LIN {X 0,Y 264.924,Z 479.026,A -85,B 0,C 180,E1 5571.318,E2 5571.318} C_VEL
LIN {X 0,Y 262.769,Z 475.669,A -85,B 0,C 180,E1 5567.921,E2 5567.921} C_VEL
LIN {X 0,Y 260.3,Z 472.231,A -85,B 0,C 180,E1 5561.41,E2 5561.41} C_VEL
LIN {X 0,Y 259.822,Z 472.519,A -85,B 0,C 180,E1 5558.558,E2 5558.558} C_VEL
LIN {X 0,Y 260.217,Z 475.555,A -85,B 0,C 180,E1 5552.295,E2 5552.295} C_VEL
LIN {X 0,Y 261.348,Z 479.248,A -85,B 0,C 180,E1 5548.559,E2 5548.559} C_VEL
LIN {X 0,Y 263.196,Z 484.586,A -85,B 0,C 180,E1 5544.765,E2 5544.765} C_VEL
LIN {X 0,Y 264.928,Z 489.758,A -85,B 0,C 180,E1 5542.035,E2 5542.035} C_VEL
LIN {X 0,Y 245.651,Z 644.406,A -85,B 0,C 180,E1 5539.399,E2 5539.399} C_VEL
LIN {X 0,Y 240.991,Z 667.184,A -85,B 0,C 180,E1 5538.834,E2 5538.834} C_VEL
LIN {X 0,Y 234.844,Z 688.807,A -85,B 0,C 180,E1 5538.055,E2 5538.055} C_VEL
LIN {X 0,Y 227.496,Z 709.005,A -85,B 0,C 180,E1 5537.061,E2 5537.061} C_VEL
LIN {X 0,Y 218.924,Z 728.293,A -85,B 0,C 180,E1 5535.814,E2 5535.814} C_VEL
LIN {X 0,Y 208.737,Z 747.497,A -85,B 0,C 180,E1 5534.186,E2 5534.186} C_VEL
LIN {X 0,Y 197.582,Z 765.406,A -85,B 0,C 180,E1 5532.183,E2 5532.183} C_VEL
LIN {X 0,Y 185.926,Z 781.624,A -85,B 0,C 180,E1 5529.792,E2 5529.792} C_VEL
LIN {X 0,Y 173.527,Z 796.762,A -85,B 0,C 180,E1 5526.82,E2 5526.82} C_VEL
LIN {X 0,Y 160.818,Z 810.467,A -85,B 0,C 180,E1 5523.174,E2 5523.174} C_VEL
LIN {X 0,Y 148.028,Z 822.753,A -85,B 0,C 180,E1 5518.662,E2 5518.662} C_VEL
LIN {X 0,Y 135.541,Z 833.645,A -85,B 0,C 180,E1 5513.019,E2 5513.019} C_VEL
LIN {X 0,Y 123.855,Z 843.086,A -85,B 0,C 180,E1 5505.936,E2 5505.936} C_VEL
LIN {X 0,Y 113.661,Z 850.993,A -85,B 0,C 180,E1 5497.079,E2 5497.079} C_VEL
LIN {X 0,Y 106.489,Z 856.756,A -85,B 0,C 180,E1 5487.315,E2 5487.315} C_VEL
LIN {X 0,Y 102.112,Z 860.954,A -85,B 0,C 180,E1 5476.414,E2 5476.414} C_VEL
LIN {X 0,Y 100.7,Z 863.459,A -85,B 0,C 180,E1 5465.36,E2 5465.36} C_VEL
LIN {X 0,Y 102.038,Z 864.682,A -85,B 0,C 180,E1 5453.997,E2 5453.997} C_VEL
LIN {X 0,Y 106.472,Z 864.54,A -85,B 0,C 180,E1 5442.914,E2 5442.914} C_VEL
LIN {X 0,Y 114.777,Z 862.689,A -85,B 0,C 180,E1 5432.097,E2 5432.097} C_VEL
LIN {X 0,Y 126.409,Z 858.943,A -85,B 0,C 180,E1 5422.802,E2 5422.802} C_VEL
LIN {X 0,Y 140.031,Z 853.547,A -85,B 0,C 180,E1 5415.453,E2 5415.453} C_VEL
LIN {X 0,Y 155.125,Z 846.474,A -85,B 0,C 180,E1 5409.569,E2 5409.569} C_VEL
LIN {X 0,Y 170.618,Z 838.065,A -85,B 0,C 180,E1 5405.018,E2 5405.018} C_VEL
LIN {X 0,Y 187.128,Z 827.692,A -85,B 0,C 180,E1 5401.224,E2 5401.224} C_VEL
LIN {X 0,Y 203.05,Z 816.054,A -85,B 0,C 180,E1 5398.276,E2 5398.276} C_VEL
LIN {X 0,Y 219.202,Z 802.456,A -85,B 0,C 180,E1 5395.814,E2 5395.814} C_VEL
LIN {X 0,Y 230.335,Z 791.931,A -85,B 0,C 180,E1 5394.32,E2 5394.32} C_VEL
LIN {X 0,Y 217.485,Z 805.371,A -85,B 0,C 180,E1 5392.785,E2 5392.785} C_VEL
LIN {X 0,Y 211.97,Z 810.64,A -85,B 0,C 180,E1 5392.344,E2 5392.344} C_VEL
LIN {X 0,Y 196.504,Z 823.434,A -85,B 0,C 180,E1 5391.994,E2 5391.994} C_VEL
LIN {X 0,Y 190.608,Z 828.015,A -85,B 0,C 180,E1 5391.411,E2 5391.411} C_VEL
LIN {X 0,Y 172.647,Z 841.576,A -85,B 0,C 180,E1 5388.143,E2 5388.143} C_VEL
LIN {X 0,Y 154.151,Z 853.984,A -85,B 0,C 180,E1 5383.715,E2 5383.715} C_VEL
LIN {X 0,Y 136.857,Z 864.412,A -85,B 0,C 180,E1 5378.088,E2 5378.088} C_VEL
LIN {X 0,Y 119.902,Z 873.894,A -85,B 0,C 180,E1 5370.13,E2 5370.13} C_VEL
LIN {X 0,Y 106.273,Z 881.294,A -85,B 0,C 180,E1 5360.223,E2 5360.223} C_VEL
LIN {X 0,Y 96.274,Z 886.967,A -85,B 0,C 180,E1 5347.78,E2 5347.78} C_VEL
LIN {X 0,Y 91.172,Z 890.787,A -85,B 0,C 180,E1 5333.932,E2 5333.932} C_VEL
LIN {X 0,Y 90.418,Z 892.658,A -85,B 0,C 180,E1 5322.122,E2 5322.122} C_VEL
LIN {X 0,Y 91.401,Z 893.227,A -85,B 0,C 180,E1 5312.501,E2 5312.501} C_VEL
LIN {X 0,Y 91.492,Z 893.013,A -85,B 0,C 180,E1 5308.115,E2 5308.115} C_VEL
LIN {X 0,Y 90.677,Z 891.796,A -85,B 0,C 180,E1 5299.832,E2 5299.832} C_VEL
LIN {X 0,Y 90.991,Z 889.004,A -85,B 0,C 180,E1 5288.732,E2 5288.732} C_VEL
LIN {X 0,Y 94.671,Z 884.089,A -85,B 0,C 180,E1 5275.954,E2 5275.954} C_VEL
LIN {X 0,Y 102.103,Z 877.465,A -85,B 0,C 180,E1 5264.36,E2 5264.36} C_VEL
LIN {X 0,Y 112.661,Z 868.974,A -85,B 0,C 180,E1 5254.612,E2 5254.612} C_VEL
LIN {X 0,Y 125.433,Z 858.784,A -85,B 0,C 180,E1 5246.767,E2 5246.767} C_VEL
LIN {X 0,Y 139.021,Z 847.405,A -85,B 0,C 180,E1 5240.766,E2 5240.766} C_VEL
LIN {X 0,Y 152.982,Z 834.686,A -85,B 0,C 180,E1 5236.092,E2 5236.092} C_VEL
LIN {X 0,Y 166.885,Z 820.612,A -85,B 0,C 180,E1 5232.41,E2 5232.41} C_VEL
LIN {X 0,Y 181.361,Z 804.213,A -85,B 0,C 180,E1 5229.289,E2 5229.289} C_VEL
LIN {X 0,Y 194.407,Z 787.495,A -85,B 0,C 180,E1 5226.945,E2 5226.945} C_VEL
LIN {X 0,Y 206.775,Z 769.259,A -85,B 0,C 180,E1 5225.031,E2 5225.031} C_VEL
LIN {X 0,Y 217.89,Z 750.129,A -85,B 0,C 180,E1 5223.53,E2 5223.53} C_VEL
LIN {X 0,Y 227.761,Z 730.153,A -85,B 0,C 180,E1 5222.336,E2 5222.336} C_VEL
LIN {X 0,Y 236.047,Z 710.089,A -85,B 0,C 180,E1 5221.423,E2 5221.423} C_VEL
LIN {X 0,Y 243.124,Z 688.824,A -85,B 0,C 180,E1 5220.708,E2 5220.708} C_VEL
LIN {X 0,Y 248.536,Z 667.243,A -85,B 0,C 180,E1 5220.164,E2 5220.164} C_VEL
LIN {X 0,Y 252.392,Z 644.573,A -85,B 0,C 180,E1 5219.681,E2 5219.681} C_VEL
LIN {X 0,Y 268.872,Z 495.81,A -85,B 0,C 180,E1 5217.075,E2 5217.075} C_VEL
LIN {X 0,Y 265.37,Z 489.707,A -85,B 0,C 180,E1 5213.293,E2 5213.293} C_VEL
LIN {X 0,Y 263.21,Z 486.145,A -85,B 0,C 180,E1 5210.379,E2 5210.379} C_VEL
LIN {X 0,Y 261.553,Z 483.485,A -85,B 0,C 180,E1 5207.64,E2 5207.64} C_VEL
LIN {X 0,Y 259.228,Z 480.152,A -85,B 0,C 180,E1 5201.33,E2 5201.33} C_VEL
LIN {X 0,Y 258.771,Z 480.458,A -85,B 0,C 180,E1 5198.626,E2 5198.626} C_VEL
LIN {X 0,Y 259.064,Z 483.366,A -85,B 0,C 180,E1 5192.588,E2 5192.588} C_VEL
LIN {X 0,Y 260.111,Z 487.05,A -85,B 0,C 180,E1 5188.869,E2 5188.869} C_VEL
LIN {X 0,Y 261.88,Z 492.466,A -85,B 0,C 180,E1 5185.063,E2 5185.063} C_VEL
LIN {X 0,Y 262.658,Z 495.183,A -85,B 0,C 180,E1 5183.653,E2 5183.653} C_VEL
LIN {X 0,Y 243.721,Z 644.757,A -85,B 0,C 180,E1 5181.215,E2 5181.215} C_VEL
LIN {X 0,Y 238.965,Z 667.665,A -85,B 0,C 180,E1 5180.679,E2 5180.679} C_VEL
LIN {X 0,Y 232.82,Z 688.959,A -85,B 0,C 180,E1 5179.955,E2 5179.955} C_VEL
LIN {X 0,Y 225.732,Z 708.262,A -85,B 0,C 180,E1 5179.066,E2 5179.066} C_VEL
LIN {X 0,Y 217.008,Z 727.792,A -85,B 0,C 180,E1 5177.889,E2 5177.889} C_VEL
LIN {X 0,Y 206.604,Z 747.209,A -85,B 0,C 180,E1 5176.348,E2 5176.348} C_VEL
LIN {X 0,Y 195.457,Z 764.898,A -85,B 0,C 180,E1 5174.497,E2 5174.497} C_VEL
LIN {X 0,Y 183.8,Z 780.948,A -85,B 0,C 180,E1 5172.285,E2 5172.285} C_VEL
LIN {X 0,Y 170.429,Z 796.941,A -85,B 0,C 180,E1 5169.321,E2 5169.321} C_VEL
LIN {X 0,Y 156.454,Z 811.547,A -85,B 0,C 180,E1 5165.564,E2 5165.564} C_VEL
LIN {X 0,Y 143.158,Z 823.823,A -85,B 0,C 180,E1 5161.125,E2 5161.125} C_VEL
LIN {X 0,Y 130.079,Z 834.717,A -85,B 0,C 180,E1 5155.501,E2 5155.501} C_VEL
LIN {X 0,Y 117.721,Z 844.169,A -85,B 0,C 180,E1 5148.321,E2 5148.321} C_VEL
LIN {X 0,Y 106.822,Z 852.097,A -85,B 0,C 180,E1 5139.161,E2 5139.161} C_VEL
LIN {X 0,Y 99.005,Z 857.931,A -85,B 0,C 180,E1 5128.749,E2 5128.749} C_VEL
LIN {X 0,Y 94.293,Z 862.111,A -85,B 0,C 180,E1 5117.14,E2 5117.14} C_VEL
LIN {X 0,Y 92.784,Z 864.707,A -85,B 0,C 180,E1 5104.844,E2 5104.844} C_VEL
LIN {X 0,Y 94.523,Z 865.971,A -85,B 0,C 180,E1 5092.164,E2 5092.164} C_VEL
LIN {X 0,Y 100.084,Z 865.743,A -85,B 0,C 180,E1 5079.724,E2 5079.724} C_VEL
LIN {X 0,Y 109.422,Z 863.853,A -85,B 0,C 180,E1 5068.705,E2 5068.705} C_VEL
LIN {X 0,Y 122.723,Z 859.924,A -85,B 0,C 180,E1 5059.093,E2 5059.093} C_VEL
LIN {X 0,Y 138.062,Z 854.158,A -85,B 0,C 180,E1 5051.698,E2 5051.698} C_VEL
LIN {X 0,Y 153.872,Z 847.013,A -85,B 0,C 180,E1 5046.222,E2 5046.222} C_VEL
LIN {X 0,Y 171.044,Z 837.891,A -85,B 0,C 180,E1 5041.755,E2 5041.755} C_VEL
LIN {X 0,Y 188.042,Z 827.35,A -85,B 0,C 180,E1 5038.317,E2 5038.317} C_VEL
LIN {X 0,Y 204.551,Z 815.529,A -85,B 0,C 180,E1 5035.637,E2 5035.637} C_VEL
LIN {X 0,Y 212.569,Z 809.08,A -85,B 0,C 180,E1 5034.476,E2 5034.476} C_VEL
LIN {X 0,Y 194.827,Z 824.66,A -85,B 0,C 180,E1 5032.062,E2 5032.062} C_VEL
LIN {X 0,Y 190.608,Z 828.015,A -85,B 0,C 180,E1 5031.411,E2 5031.411} C_VEL
LIN {X 0,Y 184.613,Z 832.571,A -85,B 0,C 180,E1 5030.763,E2 5030.763} C_VEL
LIN {X 0,Y 167.913,Z 843.389,A -85,B 0,C 180,E1 5029.908,E2 5029.908} C_VEL
LIN {X 0,Y 161.675,Z 847.223,A -85,B 0,C 180,E1 5029.028,E2 5029.028} C_VEL
LIN {X 0,Y 143.216,Z 858.371,A -85,B 0,C 180,E1 5024.441,E2 5024.441} C_VEL
LIN {X 0,Y 125.798,Z 867.854,A -85,B 0,C 180,E1 5018.409,E2 5018.409} C_VEL
LIN {X 0,Y 108.839,Z 876.387,A -85,B 0,C 180,E1 5009.704,E2 5009.704} C_VEL
LIN {X 0,Y 95.154,Z 883.089,A -85,B 0,C 180,E1 4998.24,E2 4998.24} C_VEL
LIN {X 0,Y 86.048,Z 887.879,A -85,B 0,C 180,E1 4983.892,E2 4983.892} C_VEL
LIN {X 0,Y 82.521,Z 890.822,A -85,B 0,C 180,E1 4968.355,E2 4968.355} C_VEL
LIN {X 0,Y 82.917,Z 891.818,A -85,B 0,C 180,E1 4956.919,E2 4956.919} C_VEL
LIN {X 0,Y 83.645,Z 891.917,A -85,B 0,C 180,E1 4950.678,E2 4950.678} C_VEL
LIN {X 0,Y 83.244,Z 891.408,A -85,B 0,C 180,E1 4945.17,E2 4945.17} C_VEL
LIN {X 0,Y 82.619,Z 889.427,A -85,B 0,C 180,E1 4933.831,E2 4933.831} C_VEL
LIN {X 0,Y 84.837,Z 885.454,A -85,B 0,C 180,E1 4920.323,E2 4920.323} C_VEL
LIN {X 0,Y 91.208,Z 879.636,A -85,B 0,C 180,E1 4907.174,E2 4907.174} C_VEL
LIN {X 0,Y 101.336,Z 871.983,A -85,B 0,C 180,E1 4895.985,E2 4895.985} C_VEL
LIN {X 0,Y 113.698,Z 862.812,A -85,B 0,C 180,E1 4887.343,E2 4887.343} C_VEL
LIN {X 0,Y 128.049,Z 851.724,A -85,B 0,C 180,E1 4880.434,E2 4880.434} C_VEL
LIN {X 0,Y 142.121,Z 839.968,A -85,B 0,C 180,E1 4875.444,E2 4875.444} C_VEL
LIN {X 0,Y 157.053,Z 826.029,A -85,B 0,C 180,E1 4871.34,E2 4871.34} C_VEL
LIN {X 0,Y 171.251,Z 811.205,A -85,B 0,C 180,E1 4868.237,E2 4868.237} C_VEL
LIN {X 0,Y 184.915,Z 795.071,A -85,B 0,C 180,E1 4865.759,E2 4865.759} C_VEL
LIN {X 0,Y 197.893,Z 777.601,A -85,B 0,C 180,E1 4863.767,E2 4863.767} C_VEL
LIN {X 0,Y 210.125,Z 758.395,A -85,B 0,C 180,E1 4862.142,E2 4862.142} C_VEL
LIN {X 0,Y 220.505,Z 739.281,A -85,B 0,C 180,E1 4860.924,E2 4860.924} C_VEL
LIN {X 0,Y 229.975,Z 718.523,A -85,B 0,C 180,E1 4859.917,E2 4859.917} C_VEL
LIN {X 0,Y 237.749,Z 697.676,A -85,B 0,C 180,E1 4859.159,E2 4859.159} C_VEL
LIN {X 0,Y 244.16,Z 675.65,A -85,B 0,C 180,E1 4858.583,E2 4858.583} C_VEL
LIN {X 0,Y 248.634,Z 653.809,A -85,B 0,C 180,E1 4858.117,E2 4858.117} C_VEL
LIN {X 0,Y 252.545,Z 622.713,A -85,B 0,C 180,E1 4857.551,E2 4857.551} C_VEL
LIN {X 0,Y 266.177,Z 501.282,A -85,B 0,C 180,E1 4855.476,E2 4855.476} C_VEL
LIN {X 0,Y 262.802,Z 495.248,A -85,B 0,C 180,E1 4851.358,E2 4851.358} C_VEL
LIN {X 0,Y 260.324,Z 491.281,A -85,B 0,C 180,E1 4847.316,E2 4847.316} C_VEL
LIN {X 0,Y 258.108,Z 488.034,A -85,B 0,C 180,E1 4841.011,E2 4841.011} C_VEL
LIN {X 0,Y 257.674,Z 488.539,A -85,B 0,C 180,E1 4838.37,E2 4838.37} C_VEL
LIN {X 0,Y 257.936,Z 491.276,A -85,B 0,C 180,E1 4832.781,E2 4832.781} C_VEL
LIN {X 0,Y 258.868,Z 494.803,A -85,B 0,C 180,E1 4829.219,E2 4829.219} C_VEL
LIN {X 0,Y 260.591,Z 500.432,A -85,B 0,C 180,E1 4825.307,E2 4825.307} C_VEL
LIN {X 0,Y 242.039,Z 645.097,A -85,B 0,C 180,E1 4823.058,E2 4823.058} C_VEL
LIN {X 0,Y 237.236,Z 667.943,A -85,B 0,C 180,E1 4822.557,E2 4822.557} C_VEL
LIN {X 0,Y 231.001,Z 689.276,A -85,B 0,C 180,E1 4821.88,E2 4821.88} C_VEL
LIN {X 0,Y 223.75,Z 708.751,A -85,B 0,C 180,E1 4821.039,E2 4821.039} C_VEL
LIN {X 0,Y 214.918,Z 728.218,A -85,B 0,C 180,E1 4819.937,E2 4819.937} C_VEL
LIN {X 0,Y 204.311,Z 747.686,A -85,B 0,C 180,E1 4818.486,E2 4818.486} C_VEL
LIN {X 0,Y 192.923,Z 765.427,A -85,B 0,C 180,E1 4816.737,E2 4816.737} C_VEL
LIN {X 0,Y 180.826,Z 781.713,A -85,B 0,C 180,E1 4814.61,E2 4814.61} C_VEL
LIN {X 0,Y 167.663,Z 797.067,A -85,B 0,C 180,E1 4811.91,E2 4811.91} C_VEL
LIN {X 0,Y 154.039,Z 810.974,A -85,B 0,C 180,E1 4808.549,E2 4808.549} C_VEL
LIN {X 0,Y 140.15,Z 823.513,A -85,B 0,C 180,E1 4804.31,E2 4804.31} C_VEL
LIN {X 0,Y 126.344,Z 834.65,A -85,B 0,C 180,E1 4798.87,E2 4798.87} C_VEL
LIN {X 0,Y 113.768,Z 843.888,A -85,B 0,C 180,E1 4792.21,E2 4792.21} C_VEL
LIN {X 0,Y 102.276,Z 851.801,A -85,B 0,C 180,E1 4783.575,E2 4783.575} C_VEL
LIN {X 0,Y 92.852,Z 858.206,A -85,B 0,C 180,E1 4772.475,E2 4772.475} C_VEL
LIN {X 0,Y 87.076,Z 862.639,A -85,B 0,C 180,E1 4760.089,E2 4760.089} C_VEL
LIN {X 0,Y 84.882,Z 865.617,A -85,B 0,C 180,E1 4746.398,E2 4746.398} C_VEL
LIN {X 0,Y 86.311,Z 867.154,A -85,B 0,C 180,E1 4732.968,E2 4732.968} C_VEL
LIN {X 0,Y 92.123,Z 867.233,A -85,B 0,C 180,E1 4719.01,E2 4719.01} C_VEL
LIN {X 0,Y 102.131,Z 865.538,A -85,B 0,C 180,E1 4707.029,E2 4707.029} C_VEL
LIN {X 0,Y 114.93,Z 862.236,A -85,B 0,C 180,E1 4697.725,E2 4697.725} C_VEL
LIN {X 0,Y 130.963,Z 856.914,A -85,B 0,C 180,E1 4690.009,E2 4690.009} C_VEL
LIN {X 0,Y 147.407,Z 850.224,A -85,B 0,C 180,E1 4684.43,E2 4684.43} C_VEL
LIN {X 0,Y 165.041,Z 841.662,A -85,B 0,C 180,E1 4679.999,E2 4679.999} C_VEL
LIN {X 0,Y 183.309,Z 831.088,A -85,B 0,C 180,E1 4676.471,E2 4676.471} C_VEL
LIN {X 0,Y 194.812,Z 823.518,A -85,B 0,C 180,E1 4674.64,E2 4674.64} C_VEL
LIN {X 0,Y 176.42,Z 837.275,A -85,B 0,C 180,E1 4671.853,E2 4671.853} C_VEL
LIN {X 0,Y 161.675,Z 847.223,A -85,B 0,C 180,E1 4669.028,E2 4669.028} C_VEL
LIN {X 0,Y 155.355,Z 850.938,A -85,B 0,C 180,E1 4668.048,E2 4668.048} C_VEL
LIN {X 0,Y 137.751,Z 859.678,A -85,B 0,C 180,E1 4666.353,E2 4666.353} C_VEL
LIN {X 0,Y 131.433,Z 862.733,A -85,B 0,C 180,E1 4664.999,E2 4664.999} C_VEL
LIN {X 0,Y 113.155,Z 871.566,A -85,B 0,C 180,E1 4658.078,E2 4658.078} C_VEL
LIN {X 0,Y 96.2,Z 879.117,A -85,B 0,C 180,E1 4647.988,E2 4647.988} C_VEL
LIN {X 0,Y 83.559,Z 884.671,A -85,B 0,C 180,E1 4634.899,E2 4634.899} C_VEL
LIN {X 0,Y 76.237,Z 888.317,A -85,B 0,C 180,E1 4619.02,E2 4619.02} C_VEL
LIN {X 0,Y 74.53,Z 890.286,A -85,B 0,C 180,E1 4603.175,E2 4603.175} C_VEL
LIN {X 0,Y 75.67,Z 890.639,A -85,B 0,C 180,E1 4591.506,E2 4591.506} C_VEL
LIN {X 0,Y 75.533,Z 890.311,A -85,B 0,C 180,E1 4586.957,E2 4586.957} C_VEL
LIN {X 0,Y 74.687,Z 888.722,A -85,B 0,C 180,E1 4576.048,E2 4576.048} C_VEL
LIN {X 0,Y 76.508,Z 885.109,A -85,B 0,C 180,E1 4561.075,E2 4561.075} C_VEL
LIN {X 0,Y 82.494,Z 879.907,A -85,B 0,C 180,E1 4547.245,E2 4547.245} C_VEL
LIN {X 0,Y 92.817,Z 872.605,A -85,B 0,C 180,E1 4535.035,E2 4535.035} C_VEL
LIN {X 0,Y 106.281,Z 863.376,A -85,B 0,C 180,E1 4525.415,E2 4525.415} C_VEL
LIN {X 0,Y 121.138,Z 852.652,A -85,B 0,C 180,E1 4518.328,E2 4518.328} C_VEL
LIN {X 0,Y 136.519,Z 840.416,A -85,B 0,C 180,E1 4513.057,E2 4513.057} C_VEL
LIN {X 0,Y 151.599,Z 826.97,A -85,B 0,C 180,E1 4509.109,E2 4509.109} C_VEL
LIN {X 0,Y 166.886,Z 811.628,A -85,B 0,C 180,E1 4505.958,E2 4505.958} C_VEL
LIN {X 0,Y 181.009,Z 795.521,A -85,B 0,C 180,E1 4503.57,E2 4503.57} C_VEL
LIN {X 0,Y 194.56,Z 777.741,A -85,B 0,C 180,E1 4501.644,E2 4501.644} C_VEL
LIN {X 0,Y 205.98,Z 760.302,A -85,B 0,C 180,E1 4500.233,E2 4500.233} C_VEL
LIN {X 0,Y 217.008,Z 740.709,A -85,B 0,C 180,E1 4499.033,E2 4499.033} C_VEL
LIN {X 0,Y 226.095,Z 721.625,A -85,B 0,C 180,E1 4498.138,E2 4498.138} C_VEL
LIN {X 0,Y 234.215,Z 700.744,A -85,B 0,C 180,E1 4497.404,E2 4497.404} C_VEL
LIN {X 0,Y 240.74,Z 679.476,A -85,B 0,C 180,E1 4496.864,E2 4496.864} C_VEL
LIN {X 0,Y 245.801,Z 656.965,A -85,B 0,C 180,E1 4496.402,E2 4496.402} C_VEL
LIN {X 0,Y 249.185,Z 633.378,A -85,B 0,C 180,E1 4495.971,E2 4495.971} C_VEL
LIN {X 0,Y 263.696,Z 507.078,A -85,B 0,C 180,E1 4493.906,E2 4493.906} C_VEL
LIN {X 0,Y 260.835,Z 501.998,A -85,B 0,C 180,E1 4490.068,E2 4490.068} C_VEL
LIN {X 0,Y 259.142,Z 499.12,A -85,B 0,C 180,E1 4487.07,E2 4487.07} C_VEL
LIN {X 0,Y 257.04,Z 495.955,A -85,B 0,C 180,E1 4480.929,E2 4480.929} C_VEL
LIN {X 0,Y 256.6,Z 496.55,A -85,B 0,C 180,E1 4478.275,E2 4478.275} C_VEL
LIN {X 0,Y 256.802,Z 499.085,A -85,B 0,C 180,E1 4473.08,E2 4473.08} C_VEL
LIN {X 0,Y 257.635,Z 502.557,A -85,B 0,C 180,E1 4469.573,E2 4469.573} C_VEL
LIN {X 0,Y 258.592,Z 506.364,A -85,B 0,C 180,E1 4466.959,E2 4466.959} C_VEL
LIN {X 0,Y 240.541,Z 645.36,A -85,B 0,C 180,E1 4464.923,E2 4464.923} C_VEL
LIN {X 0,Y 235.666,Z 668.296,A -85,B 0,C 180,E1 4464.457,E2 4464.457} C_VEL
LIN {X 0,Y 229.201,Z 690.109,A -85,B 0,C 180,E1 4463.811,E2 4463.811} C_VEL
LIN {X 0,Y 221.604,Z 710.096,A -85,B 0,C 180,E1 4463.001,E2 4463.001} C_VEL
LIN {X 0,Y 212.569,Z 729.539,A -85,B 0,C 180,E1 4461.964,E2 4461.964} C_VEL
LIN {X 0,Y 201.832,Z 748.804,A -85,B 0,C 180,E1 4460.611,E2 4460.611} C_VEL
LIN {X 0,Y 190.22,Z 766.486,A -85,B 0,C 180,E1 4458.967,E2 4458.967} C_VEL
LIN {X 0,Y 177.853,Z 782.736,A -85,B 0,C 180,E1 4456.961,E2 4456.961} C_VEL
LIN {X 0,Y 164.355,Z 798.084,A -85,B 0,C 180,E1 4454.4,E2 4454.4} C_VEL
LIN {X 0,Y 150.32,Z 811.981,A -85,B 0,C 180,E1 4451.19,E2 4451.19} C_VEL
LIN {X 0,Y 135.931,Z 824.521,A -85,B 0,C 180,E1 4447.102,E2 4447.102} C_VEL
LIN {X 0,Y 121.513,Z 835.67,A -85,B 0,C 180,E1 4441.783,E2 4441.783} C_VEL
LIN {X 0,Y 108.242,Z 844.928,A -85,B 0,C 180,E1 4435.151,E2 4435.151} C_VEL
LIN {X 0,Y 95.783,Z 852.972,A -85,B 0,C 180,E1 4426.195,E2 4426.195} C_VEL
LIN {X 0,Y 85.716,Z 859.296,A -85,B 0,C 180,E1 4414.69,E2 4414.69} C_VEL
LIN {X 0,Y 79.356,Z 863.766,A -85,B 0,C 180,E1 4401.311,E2 4401.311} C_VEL
LIN {X 0,Y 76.959,Z 866.799,A -85,B 0,C 180,E1 4386.258,E2 4386.258} C_VEL
LIN {X 0,Y 78.656,Z 868.415,A -85,B 0,C 180,E1 4371.483,E2 4371.483} C_VEL
LIN {X 0,Y 84.96,Z 868.558,A -85,B 0,C 180,E1 4356.857,E2 4356.857} C_VEL
LIN {X 0,Y 95.59,Z 867.073,A -85,B 0,C 180,E1 4344.51,E2 4344.51} C_VEL
LIN {X 0,Y 109.605,Z 863.897,A -85,B 0,C 180,E1 4334.79,E2 4334.79} C_VEL
LIN {X 0,Y 125.099,Z 859.275,A -85,B 0,C 180,E1 4327.701,E2 4327.701} C_VEL
LIN {X 0,Y 143.049,Z 852.564,A -85,B 0,C 180,E1 4321.935,E2 4321.935} C_VEL
LIN {X 0,Y 162.12,Z 843.776,A -85,B 0,C 180,E1 4317.496,E2 4317.496} C_VEL
LIN {X 0,Y 176.954,Z 835.724,A -85,B 0,C 180,E1 4314.812,E2 4314.812} C_VEL
LIN {X 0,Y 157.697,Z 848.116,A -85,B 0,C 180,E1 4311.503,E2 4311.503} C_VEL
LIN {X 0,Y 138.486,Z 859.055,A -85,B 0,C 180,E1 4307.059,E2 4307.059} C_VEL
LIN {X 0,Y 131.433,Z 862.733,A -85,B 0,C 180,E1 4304.999,E2 4304.999} C_VEL
LIN {X 0,Y 125.109,Z 865.686,A -85,B 0,C 180,E1 4303.476,E2 4303.476} C_VEL
LIN {X 0,Y 106.282,Z 872.566,A -85,B 0,C 180,E1 4299.946,E2 4299.946} C_VEL
LIN {X 0,Y 101.047,Z 874.438,A -85,B 0,C 180,E1 4297.94,E2 4297.94} C_VEL
LIN {X 0,Y 84.154,Z 881.038,A -85,B 0,C 180,E1 4286.259,E2 4286.259} C_VEL
LIN {X 0,Y 72.286,Z 885.684,A -85,B 0,C 180,E1 4270.538,E2 4270.538} C_VEL
LIN {X 0,Y 66.939,Z 888.365,A -85,B 0,C 180,E1 4251.917,E2 4251.917} C_VEL
LIN {X 0,Y 67.061,Z 889.298,A -85,B 0,C 180,E1 4236.841,E2 4236.841} C_VEL
LIN {X 0,Y 67.884,Z 889.245,A -85,B 0,C 180,E1 4229.991,E2 4229.991} C_VEL
LIN {X 0,Y 66.94,Z 888.229,A -85,B 0,C 180,E1 4220.356,E2 4220.356} C_VEL
LIN {X 0,Y 67.525,Z 885.51,A -85,B 0,C 180,E1 4205.496,E2 4205.496} C_VEL
LIN {X 0,Y 72.952,Z 880.641,A -85,B 0,C 180,E1 4188.852,E2 4188.852} C_VEL
LIN {X 0,Y 83.092,Z 873.998,A -85,B 0,C 180,E1 4175.079,E2 4175.079} C_VEL
LIN {X 0,Y 96.725,Z 865.334,A -85,B 0,C 180,E1 4164.527,E2 4164.527} C_VEL
LIN {X 0,Y 111.874,Z 855.197,A -85,B 0,C 180,E1 4156.986,E2 4156.986} C_VEL
LIN {X 0,Y 127.554,Z 843.645,A -85,B 0,C 180,E1 4151.505,E2 4151.505} C_VEL
LIN {X 0,Y 143.193,Z 830.78,A -85,B 0,C 180,E1 4147.437,E2 4147.437} C_VEL
LIN {X 0,Y 159.405,Z 815.516,A -85,B 0,C 180,E1 4144.156,E2 4144.156} C_VEL
LIN {X 0,Y 173.573,Z 800.272,A -85,B 0,C 180,E1 4141.839,E2 4141.839} C_VEL
LIN {X 0,Y 187.432,Z 783.218,A -85,B 0,C 180,E1 4139.945,E2 4139.945} C_VEL
LIN {X 0,Y 200.051,Z 765.299,A -85,B 0,C 180,E1 4138.465,E2 4138.465} C_VEL
LIN {X 0,Y 211.538,Z 746.139,A -85,B 0,C 180,E1 4137.292,E2 4137.292} C_VEL
LIN {X 0,Y 221.539,Z 726.3,A -85,B 0,C 180,E1 4136.378,E2 4136.378} C_VEL
LIN {X 0,Y 230.391,Z 704.98,A -85,B 0,C 180,E1 4135.641,E2 4135.641} C_VEL
LIN {X 0,Y 237.461,Z 683.608,A -85,B 0,C 180,E1 4135.107,E2 4135.107} C_VEL
LIN {X 0,Y 242.864,Z 661.813,A -85,B 0,C 180,E1 4134.679,E2 4134.679} C_VEL
LIN {X 0,Y 246.515,Z 639.065,A -85,B 0,C 180,E1 4134.274,E2 4134.274} C_VEL
LIN {X 0,Y 261.288,Z 512.956,A -85,B 0,C 180,E1 4132.304,E2 4132.304} C_VEL
LIN {X 0,Y 259.205,Z 509.218,A -85,B 0,C 180,E1 4129.218,E2 4129.218} C_VEL
LIN {X 0,Y 257.892,Z 506.891,A -85,B 0,C 180,E1 4126.697,E2 4126.697} C_VEL
LIN {X 0,Y 255.966,Z 503.875,A -85,B 0,C 180,E1 4120.846,E2 4120.846} C_VEL
LIN {X 0,Y 255.494,Z 504.667,A -85,B 0,C 180,E1 4117.934,E2 4117.934} C_VEL
LIN {X 0,Y 255.664,Z 506.876,A -85,B 0,C 180,E1 4113.399,E2 4113.399} C_VEL
LIN {X 0,Y 256.446,Z 510.461,A -85,B 0,C 180,E1 4109.805,E2 4109.805} C_VEL
LIN {X 0,Y 256.815,Z 512.184,A -85,B 0,C 180,E1 4108.644,E2 4108.644} C_VEL
LIN {X 0,Y 239.269,Z 645.747,A -85,B 0,C 180,E1 4106.807,E2 4106.807} C_VEL
LIN {X 0,Y 234.34,Z 668.679,A -85,B 0,C 180,E1 4106.378,E2 4106.378} C_VEL
LIN {X 0,Y 227.903,Z 690.175,A -85,B 0,C 180,E1 4105.794,E2 4105.794} C_VEL
LIN {X 0,Y 220.199,Z 710.275,A -85,B 0,C 180,E1 4105.048,E2 4105.048} C_VEL
LIN {X 0,Y 211.086,Z 729.693,A -85,B 0,C 180,E1 4104.098,E2 4104.098} C_VEL
LIN {X 0,Y 200.114,Z 749.148,A -85,B 0,C 180,E1 4102.842,E2 4102.842} C_VEL
LIN {X 0,Y 188.283,Z 766.904,A -85,B 0,C 180,E1 4101.322,E2 4101.322} C_VEL
LIN {X 0,Y 175.656,Z 783.224,A -85,B 0,C 180,E1 4099.46,E2 4099.46} C_VEL
LIN {X 0,Y 161.021,Z 799.465,A -85,B 0,C 180,E1 4096.92,E2 4096.92} C_VEL
LIN {X 0,Y 146.048,Z 813.795,A -85,B 0,C 180,E1 4093.75,E2 4093.75} C_VEL
LIN {X 0,Y 131.197,Z 826.193,A -85,B 0,C 180,E1 4089.81,E2 4089.81} C_VEL
LIN {X 0,Y 116.209,Z 837.227,A -85,B 0,C 180,E1 4084.607,E2 4084.607} C_VEL
LIN {X 0,Y 101.467,Z 846.888,A -85,B 0,C 180,E1 4077.524,E2 4077.524} C_VEL
LIN {X 0,Y 88.436,Z 854.706,A -85,B 0,C 180,E1 4068.258,E2 4068.258} C_VEL
LIN {X 0,Y 77.807,Z 860.944,A -85,B 0,C 180,E1 4055.908,E2 4055.908} C_VEL
LIN {X 0,Y 70.956,Z 865.501,A -85,B 0,C 180,E1 4040.273,E2 4040.273} C_VEL
LIN {X 0,Y 69.043,Z 868.267,A -85,B 0,C 180,E1 4023.871,E2 4023.871} C_VEL
LIN {X 0,Y 71.85,Z 869.761,A -85,B 0,C 180,E1 4007.021,E2 4007.021} C_VEL
LIN {X 0,Y 79.832,Z 869.809,A -85,B 0,C 180,E1 3991.622,E2 3991.622} C_VEL
LIN {X 0,Y 92.91,Z 868.049,A -85,B 0,C 180,E1 3978.756,E2 3978.756} C_VEL
LIN {X 0,Y 108.795,Z 864.526,A -85,B 0,C 180,E1 3969.52,E2 3969.52} C_VEL
LIN {X 0,Y 126.131,Z 859.396,A -85,B 0,C 180,E1 3962.889,E2 3962.889} C_VEL
LIN {X 0,Y 145.072,Z 852.341,A -85,B 0,C 180,E1 3957.826,E2 3957.826} C_VEL
LIN {X 0,Y 158.956,Z 846.171,A -85,B 0,C 180,E1 3954.957,E2 3954.957} C_VEL
LIN {X 0,Y 138.687,Z 857.351,A -85,B 0,C 180,E1 3950.971,E2 3950.971} C_VEL
LIN {X 0,Y 118.72,Z 866.947,A -85,B 0,C 180,E1 3945.363,E2 3945.363} C_VEL
LIN {X 0,Y 101.047,Z 874.438,A -85,B 0,C 180,E1 3937.94,E2 3937.94} C_VEL
LIN {X 0,Y 95.006,Z 876.599,A -85,B 0,C 180,E1 3935.36,E2 3935.36} C_VEL
LIN {X 0,Y 77.172,Z 881.073,A -85,B 0,C 180,E1 3928.228,E2 3928.228} C_VEL
LIN {X 0,Y 72.703,Z 882.264,A -85,B 0,C 180,E1 3924.553,E2 3924.553} C_VEL
LIN {X 0,Y 62.088,Z 885.88,A -85,B 0,C 180,E1 3906.366,E2 3906.366} C_VEL
LIN {X 0,Y 58.667,Z 887.692,A -85,B 0,C 180,E1 3885.813,E2 3885.813} C_VEL
LIN {X 0,Y 59.752,Z 887.979,A -85,B 0,C 180,E1 3871.908,E2 3871.908} C_VEL
LIN {X 0,Y 59.9,Z 887.866,A -85,B 0,C 180,E1 3869.034,E2 3869.034} C_VEL
LIN {X 0,Y 58.841,Z 886.347,A -85,B 0,C 180,E1 3855.611,E2 3855.611} C_VEL
LIN {X 0,Y 61.506,Z 882.676,A -85,B 0,C 180,E1 3836.435,E2 3836.435} C_VEL
LIN {X 0,Y 69.367,Z 877.45,A -85,B 0,C 180,E1 3820.175,E2 3820.175} C_VEL
LIN {X 0,Y 81.298,Z 870.497,A -85,B 0,C 180,E1 3807.672,E2 3807.672} C_VEL
LIN {X 0,Y 95.945,Z 861.804,A -85,B 0,C 180,E1 3798.483,E2 3798.483} C_VEL
LIN {X 0,Y 112.348,Z 851.174,A -85,B 0,C 180,E1 3791.752,E2 3791.752} C_VEL
LIN {X 0,Y 128.939,Z 838.976,A -85,B 0,C 180,E1 3786.954,E2 3786.954} C_VEL
LIN {X 0,Y 144.378,Z 826.11,A -85,B 0,C 180,E1 3783.575,E2 3783.575} C_VEL
LIN {X 0,Y 160.005,Z 811.336,A -85,B 0,C 180,E1 3780.892,E2 3780.892} C_VEL
LIN {X 0,Y 175.022,Z 795.042,A -85,B 0,C 180,E1 3778.791,E2 3778.791} C_VEL
LIN {X 0,Y 189.218,Z 777.088,A -85,B 0,C 180,E1 3777.136,E2 3777.136} C_VEL
LIN {X 0,Y 201.494,Z 758.977,A -85,B 0,C 180,E1 3775.903,E2 3775.903} C_VEL
LIN {X 0,Y 213.088,Z 738.824,A -85,B 0,C 180,E1 3774.886,E2 3774.886} C_VEL
LIN {X 0,Y 222.511,Z 719.245,A -85,B 0,C 180,E1 3774.139,E2 3774.139} C_VEL
LIN {X 0,Y 230.852,Z 698.052,A -85,B 0,C 180,E1 3773.535,E2 3773.535} C_VEL
LIN {X 0,Y 237.672,Z 675.638,A -85,B 0,C 180,E1 3773.085,E2 3773.085} C_VEL
LIN {X 0,Y 242.357,Z 654.189,A -85,B 0,C 180,E1 3772.708,E2 3772.708} C_VEL
LIN {X 0,Y 246.352,Z 625.13,A -85,B 0,C 180,E1 3772.241,E2 3772.241} C_VEL
LIN {X 0,Y 259.041,Z 518.92,A -85,B 0,C 180,E1 3770.615,E2 3770.615} C_VEL
LIN {X 0,Y 256.843,Z 514.875,A -85,B 0,C 180,E1 3766.717,E2 3766.717} C_VEL
LIN {X 0,Y 254.891,Z 511.795,A -85,B 0,C 180,E1 3760.762,E2 3760.762} C_VEL
LIN {X 0,Y 254.395,Z 512.786,A -85,B 0,C 180,E1 3757.59,E2 3757.59} C_VEL
LIN {X 0,Y 254.549,Z 514.795,A -85,B 0,C 180,E1 3753.586,E2 3753.586} C_VEL
LIN {X 0,Y 255.172,Z 518.003,A -85,B 0,C 180,E1 3750.35,E2 3750.35} C_VEL
LIN {X 0,Y 238.189,Z 646.072,A -85,B 0,C 180,E1 3748.709,E2 3748.709} C_VEL
LIN {X 0,Y 233.235,Z 668.928,A -85,B 0,C 180,E1 3748.319,E2 3748.319} C_VEL
LIN {X 0,Y 226.631,Z 690.766,A -85,B 0,C 180,E1 3747.78,E2 3747.78} C_VEL
LIN {X 0,Y 219.07,Z 710.28,A -85,B 0,C 180,E1 3747.122,E2 3747.122} C_VEL
LIN {X 0,Y 209.833,Z 729.817,A -85,B 0,C 180,E1 3746.257,E2 3746.257} C_VEL
LIN {X 0,Y 199.179,Z 748.606,A -85,B 0,C 180,E1 3745.165,E2 3745.165} C_VEL
LIN {X 0,Y 187.145,Z 766.577,A -85,B 0,C 180,E1 3743.784,E2 3743.784} C_VEL
LIN {X 0,Y 173.791,Z 783.604,A -85,B 0,C 180,E1 3742.021,E2 3742.021} C_VEL
LIN {X 0,Y 159.181,Z 799.533,A -85,B 0,C 180,E1 3739.75,E2 3739.75} C_VEL
LIN {X 0,Y 144.818,Z 813.085,A -85,B 0,C 180,E1 3737.047,E2 3737.047} C_VEL
LIN {X 0,Y 129.434,Z 825.772,A -85,B 0,C 180,E1 3733.439,E2 3733.439} C_VEL
LIN {X 0,Y 113.751,Z 837.074,A -85,B 0,C 180,E1 3728.621,E2 3728.621} C_VEL
LIN {X 0,Y 98.969,Z 846.494,A -85,B 0,C 180,E1 3722.381,E2 3722.381} C_VEL
LIN {X 0,Y 84.123,Z 854.926,A -85,B 0,C 180,E1 3713.1,E2 3713.1} C_VEL
LIN {X 0,Y 72.297,Z 861.212,A -85,B 0,C 180,E1 3700.93,E2 3700.93} C_VEL
LIN {X 0,Y 64.061,Z 865.991,A -85,B 0,C 180,E1 3684.636,E2 3684.636} C_VEL
LIN {X 0,Y 61.113,Z 869.155,A -85,B 0,C 180,E1 3665.868,E2 3665.868} C_VEL
LIN {X 0,Y 63.555,Z 870.891,A -85,B 0,C 180,E1 3647.444,E2 3647.444} C_VEL
LIN {X 0,Y 72.01,Z 871.188,A -85,B 0,C 180,E1 3629.987,E2 3629.987} C_VEL
LIN {X 0,Y 85.512,Z 869.823,A -85,B 0,C 180,E1 3616.531,E2 3616.531} C_VEL
LIN {X 0,Y 102.867,Z 866.567,A -85,B 0,C 180,E1 3606.696,E2 3606.696} C_VEL
LIN {X 0,Y 120.972,Z 861.797,A -85,B 0,C 180,E1 3600.171,E2 3600.171} C_VEL
LIN {X 0,Y 140.433,Z 855.159,A -85,B 0,C 180,E1 3595.335,E2 3595.335} C_VEL
LIN {X 0,Y 141.066,Z 854.928,A -85,B 0,C 180,E1 3595.137,E2 3595.137} C_VEL
LIN {X 0,Y 120.457,Z 864.495,A -85,B 0,C 180,E1 3590.442,E2 3590.442} C_VEL
LIN {X 0,Y 100.129,Z 872.706,A -85,B 0,C 180,E1 3583.438,E2 3583.438} C_VEL
LIN {X 0,Y 81.881,Z 879.227,A -85,B 0,C 180,E1 3573.034,E2 3573.034} C_VEL
LIN {X 0,Y 72.703,Z 882.264,A -85,B 0,C 180,E1 3564.553,E2 3564.553} C_VEL
LIN {X 0,Y 67.785,Z 883.509,A -85,B 0,C 180,E1 3559.741,E2 3559.741} C_VEL
LIN {X 0,Y 53.959,Z 885.436,A -85,B 0,C 180,E1 3544.469,E2 3544.469} C_VEL
LIN {X 0,Y 51.718,Z 885.908,A -85,B 0,C 180,E1 3537.656,E2 3537.656} C_VEL
LIN {X 0,Y 51.28,Z 886.674,A -85,B 0,C 180,E1 3516.031,E2 3516.031} C_VEL
LIN {X 0,Y 51.997,Z 886.573,A -85,B 0,C 180,E1 3509.596,E2 3509.596} C_VEL
LIN {X 0,Y 50.927,Z 884.999,A -85,B 0,C 180,E1 3494.034,E2 3494.034} C_VEL
LIN {X 0,Y 54.74,Z 881.077,A -85,B 0,C 180,E1 3471.596,E2 3471.596} C_VEL
LIN {X 0,Y 64.865,Z 875.388,A -85,B 0,C 180,E1 3453.64,E2 3453.64} C_VEL
LIN {X 0,Y 79.283,Z 867.755,A -85,B 0,C 180,E1 3441.037,E2 3441.037} C_VEL
LIN {X 0,Y 95.463,Z 858.546,A -85,B 0,C 180,E1 3432.708,E2 3432.708} C_VEL
LIN {X 0,Y 112.8,Z 847.478,A -85,B 0,C 180,E1 3426.856,E2 3426.856} C_VEL
LIN {X 0,Y 129.157,Z 835.609,A -85,B 0,C 180,E1 3422.91,E2 3422.91} C_VEL
LIN {X 0,Y 145.988,Z 821.552,A -85,B 0,C 180,E1 3419.844,E2 3419.844} C_VEL
LIN {X 0,Y 161.522,Z 806.587,A -85,B 0,C 180,E1 3417.614,E2 3417.614} C_VEL
LIN {X 0,Y 176.444,Z 789.997,A -85,B 0,C 180,E1 3415.859,E2 3415.859} C_VEL
LIN {X 0,Y 189.846,Z 772.756,A -85,B 0,C 180,E1 3414.528,E2 3414.528} C_VEL
LIN {X 0,Y 202.295,Z 754.089,A -85,B 0,C 180,E1 3413.463,E2 3413.463} C_VEL
LIN {X 0,Y 213.235,Z 734.539,A -85,B 0,C 180,E1 3412.64,E2 3412.64} C_VEL
LIN {X 0,Y 222.653,Z 714.315,A -85,B 0,C 180,E1 3411.999,E2 3411.999} C_VEL
LIN {X 0,Y 230.761,Z 692.815,A -85,B 0,C 180,E1 3411.498,E2 3411.498} C_VEL
LIN {X 0,Y 237.068,Z 671.219,A -85,B 0,C 180,E1 3411.125,E2 3411.125} C_VEL
LIN {X 0,Y 241.652,Z 649.054,A -85,B 0,C 180,E1 3410.765,E2 3410.765} C_VEL
LIN {X 0,Y 256.903,Z 525.146,A -85,B 0,C 180,E1 3408.966,E2 3408.966} C_VEL
LIN {X 0,Y 255.461,Z 522.512,A -85,B 0,C 180,E1 3406.092,E2 3406.092} C_VEL
LIN {X 0,Y 253.816,Z 519.717,A -85,B 0,C 180,E1 3400.678,E2 3400.678} C_VEL
LIN {X 0,Y 253.334,Z 521.63,A -85,B 0,C 180,E1 3395.519,E2 3395.519} C_VEL
LIN {X 0,Y 253.477,Z 523.053,A -85,B 0,C 180,E1 3393.404,E2 3393.404} C_VEL
LIN {X 0,Y 253.7,Z 524.384,A -85,B 0,C 180,E1 3392.069,E2 3392.069} C_VEL
LIN {X 0,Y 237.372,Z 646.3,A -85,B 0,C 180,E1 3390.625,E2 3390.625} C_VEL
LIN {X 0,Y 232.367,Z 669.227,A -85,B 0,C 180,E1 3390.275,E2 3390.275} C_VEL
LIN {X 0,Y 225.877,Z 690.565,A -85,B 0,C 180,E1 3389.805,E2 3389.805} C_VEL
LIN {X 0,Y 218.23,Z 710.252,A -85,B 0,C 180,E1 3389.216,E2 3389.216} C_VEL
LIN {X 0,Y 208.388,Z 730.848,A -85,B 0,C 180,E1 3388.396,E2 3388.396} C_VEL
LIN {X 0,Y 197.101,Z 750.346,A -85,B 0,C 180,E1 3387.366,E2 3387.366} C_VEL
LIN {X 0,Y 184.842,Z 768.22,A -85,B 0,C 180,E1 3386.109,E2 3386.109} C_VEL
LIN {X 0,Y 171.315,Z 785.077,A -85,B 0,C 180,E1 3384.511,E2 3384.511} C_VEL
LIN {X 0,Y 156.421,Z 800.942,A -85,B 0,C 180,E1 3382.436,E2 3382.436} C_VEL
LIN {X 0,Y 141.028,Z 815.018,A -85,B 0,C 180,E1 3379.824,E2 3379.824} C_VEL
LIN {X 0,Y 125.439,Z 827.378,A -85,B 0,C 180,E1 3376.504,E2 3376.504} C_VEL
LIN {X 0,Y 108.32,Z 839.134,A -85,B 0,C 180,E1 3371.658,E2 3371.658} C_VEL
LIN {X 0,Y 92.088,Z 848.805,A -85,B 0,C 180,E1 3365.139,E2 3365.139} C_VEL
LIN {X 0,Y 77.267,Z 856.648,A -85,B 0,C 180,E1 3356.11,E2 3356.11} C_VEL
LIN {X 0,Y 64.255,Z 863.053,A -85,B 0,C 180,E1 3342.592,E2 3342.592} C_VEL
LIN {X 0,Y 55.886,Z 867.503,A -85,B 0,C 180,E1 3324.878,E2 3324.878} C_VEL
LIN {X 0,Y 53.212,Z 870.565,A -85,B 0,C 180,E1 3303.208,E2 3303.208} C_VEL
LIN {X 0,Y 56.882,Z 872.256,A -85,B 0,C 180,E1 3282.432,E2 3282.432} C_VEL
LIN {X 0,Y 67.781,Z 872.474,A -85,B 0,C 180,E1 3263.467,E2 3263.467} C_VEL
LIN {X 0,Y 82.498,Z 871.047,A -85,B 0,C 180,E1 3251.018,E2 3251.018} C_VEL
LIN {X 0,Y 101.037,Z 867.778,A -85,B 0,C 180,E1 3242.028,E2 3242.028} C_VEL
LIN {X 0,Y 120.246,Z 862.93,A -85,B 0,C 180,E1 3236.123,E2 3236.123} C_VEL
LIN {X 0,Y 123.135,Z 862.073,A -85,B 0,C 180,E1 3235.341,E2 3235.341} C_VEL
LIN {X 0,Y 101.67,Z 870.461,A -85,B 0,C 180,E1 3229.522,E2 3229.522} C_VEL
LIN {X 0,Y 81.615,Z 877.178,A -85,B 0,C 180,E1 3220.594,E2 3220.594} C_VEL
LIN {X 0,Y 64.654,Z 882.052,A -85,B 0,C 180,E1 3206.609,E2 3206.609} C_VEL
LIN {X 0,Y 53.46,Z 885.258,A -85,B 0,C 180,E1 3185.422,E2 3185.422} C_VEL
LIN {X 0,Y 51.718,Z 885.908,A -85,B 0,C 180,E1 3177.656,E2 3177.656} C_VEL
LIN {X 0,Y 49.953,Z 886.25,A -85,B 0,C 180,E1 3169.749,E2 3169.749} C_VEL
LIN {X 0,Y 47.089,Z 886.027,A -85,B 0,C 180,E1 3159.691,E2 3159.691} C_VEL
LIN {X 0,Y 43.404,Z 884.687,A -85,B 0,C 180,E1 3142.042,E2 3142.042} C_VEL
LIN {X 0,Y 43.004,Z 883.898,A -85,B 0,C 180,E1 3134.435,E2 3134.435} C_VEL
LIN {X 0,Y 47.154,Z 880.188,A -85,B 0,C 180,E1 3108.888,E2 3108.888} C_VEL
LIN {X 0,Y 58.453,Z 874.621,A -85,B 0,C 180,E1 3089.245,E2 3089.245} C_VEL
LIN {X 0,Y 74.062,Z 867.062,A -85,B 0,C 180,E1 3076.533,E2 3076.533} C_VEL
LIN {X 0,Y 91.027,Z 858.012,A -85,B 0,C 180,E1 3068.629,E2 3068.629} C_VEL
LIN {X 0,Y 108.187,Z 847.628,A -85,B 0,C 180,E1 3063.427,E2 3063.427} C_VEL
LIN {X 0,Y 125.994,Z 835.213,A -85,B 0,C 180,E1 3059.613,E2 3059.613} C_VEL
LIN {X 0,Y 143.201,Z 821.184,A -85,B 0,C 180,E1 3056.874,E2 3056.874} C_VEL
LIN {X 0,Y 159.068,Z 806.219,A -85,B 0,C 180,E1 3054.892,E2 3054.892} C_VEL
LIN {X 0,Y 174.675,Z 789.169,A -85,B 0,C 180,E1 3053.305,E2 3053.305} C_VEL
LIN {X 0,Y 188.229,Z 771.95,A -85,B 0,C 180,E1 3052.146,E2 3052.146} C_VEL
LIN {X 0,Y 200.307,Z 754.06,A -85,B 0,C 180,E1 3051.257,E2 3051.257} C_VEL
LIN {X 0,Y 211.319,Z 734.646,A -85,B 0,C 180,E1 3050.543,E2 3050.543} C_VEL
LIN {X 0,Y 220.842,Z 714.486,A -85,B 0,C 180,E1 3049.985,E2 3049.985} C_VEL
LIN {X 0,Y 228.761,Z 693.903,A -85,B 0,C 180,E1 3049.563,E2 3049.563} C_VEL
LIN {X 0,Y 235.211,Z 672.473,A -85,B 0,C 180,E1 3049.239,E2 3049.239} C_VEL
LIN {X 0,Y 239.936,Z 650.315,A -85,B 0,C 180,E1 3048.914,E2 3048.914} C_VEL
LIN {X 0,Y 245.805,Z 605.358,A -85,B 0,C 180,E1 3048.292,E2 3048.292} C_VEL
LIN {X 0,Y 254.957,Z 531.543,A -85,B 0,C 180,E1 3047.286,E2 3047.286} C_VEL
LIN {X 0,Y 254.089,Z 530.125,A -85,B 0,C 180,E1 3045.414,E2 3045.414} C_VEL
LIN {X 0,Y 252.742,Z 527.642,A -85,B 0,C 180,E1 3040.592,E2 3040.592} C_VEL
LIN {X 0,Y 252.318,Z 530.335,A -85,B 0,C 180,E1 3034.285,E2 3034.285} C_VEL
LIN {X 0,Y 252.319,Z 531.002,A -85,B 0,C 180,E1 3033.805,E2 3033.805} C_VEL
LIN {X 0,Y 236.722,Z 646.668,A -85,B 0,C 180,E1 3032.551,E2 3032.551} C_VEL
LIN {X 0,Y 231.669,Z 669.644,A -85,B 0,C 180,E1 3032.241,E2 3032.241} C_VEL
LIN {X 0,Y 225.152,Z 690.898,A -85,B 0,C 180,E1 3031.828,E2 3031.828} C_VEL
LIN {X 0,Y 217.363,Z 710.785,A -85,B 0,C 180,E1 3031.303,E2 3031.303} C_VEL
LIN {X 0,Y 207.728,Z 730.808,A -85,B 0,C 180,E1 3030.604,E2 3030.604} C_VEL
LIN {X 0,Y 196.803,Z 749.665,A -85,B 0,C 180,E1 3029.738,E2 3029.738} C_VEL
LIN {X 0,Y 184.447,Z 767.685,A -85,B 0,C 180,E1 3028.643,E2 3028.643} C_VEL
LIN {X 0,Y 170.146,Z 785.362,A -85,B 0,C 180,E1 3027.181,E2 3027.181} C_VEL
LIN {X 0,Y 154.98,Z 801.287,A -85,B 0,C 180,E1 3025.349,E2 3025.349} C_VEL
LIN {X 0,Y 139.962,Z 814.853,A -85,B 0,C 180,E1 3023.146,E2 3023.146} C_VEL
LIN {X 0,Y 123.713,Z 827.573,A -85,B 0,C 180,E1 3020.163,E2 3020.163} C_VEL
LIN {X 0,Y 106.894,Z 838.927,A -85,B 0,C 180,E1 3016.081,E2 3016.081} C_VEL
LIN {X 0,Y 90.681,Z 848.408,A -85,B 0,C 180,E1 3010.591,E2 3010.591} C_VEL
LIN {X 0,Y 73.814,Z 856.89,A -85,B 0,C 180,E1 3001.898,E2 3001.898} C_VEL
LIN {X 0,Y 59.84,Z 863.184,A -85,B 0,C 180,E1 2989.533,E2 2989.533} C_VEL
LIN {X 0,Y 48.99,Z 868.237,A -85,B 0,C 180,E1 2969.652,E2 2969.652} C_VEL
LIN {X 0,Y 45.281,Z 871.372,A -85,B 0,C 180,E1 2946.595,E2 2946.595} C_VEL
LIN {X 0,Y 48.561,Z 873.248,A -85,B 0,C 180,E1 2922.183,E2 2922.183} C_VEL
LIN {X 0,Y 59.294,Z 873.85,A -85,B 0,C 180,E1 2901.772,E2 2901.772} C_VEL
LIN {X 0,Y 74.767,Z 872.939,A -85,B 0,C 180,E1 2888.328,E2 2888.328} C_VEL
LIN {X 0,Y 93.984,Z 870.217,A -85,B 0,C 180,E1 2879.224,E2 2879.224} C_VEL
LIN {X 0,Y 105.284,Z 867.924,A -85,B 0,C 180,E1 2875.598,E2 2875.598} C_VEL
LIN {X 0,Y 82.935,Z 875.003,A -85,B 0,C 180,E1 2868.171,E2 2868.171} C_VEL
LIN {X 0,Y 63.396,Z 880.145,A -85,B 0,C 180,E1 2856.146,E2 2856.146} C_VEL
LIN {X 0,Y 48.462,Z 883.633,A -85,B 0,C 180,E1 2835.449,E2 2835.449} C_VEL
LIN {X 0,Y 42.989,Z 885.095,A -85,B 0,C 180,E1 2810.403,E2 2810.403} C_VEL
LIN {X 0,Y 43.998,Z 885.262,A -85,B 0,C 180,E1 2790.418,E2 2790.418} C_VEL
LIN {X 0,Y 43.004,Z 883.898,A -85,B 0,C 180,E1 2774.435,E2 2774.435} C_VEL
LIN {X 0,Y 42.704,Z 882.74,A -85,B 0,C 180,E1 2764.93,E2 2764.93} C_VEL
LIN {X 0,Y 42.326,Z 880.079,A -85,B 0,C 180,E1 2748.674,E2 2748.674} C_VEL
LIN {X 0,Y 45.156,Z 877.049,A -85,B 0,C 180,E1 2734.143,E2 2734.143} C_VEL
LIN {X 0,Y 47.572,Z 875.811,A -85,B 0,C 180,E1 2729.733,E2 2729.733} C_VEL
LIN {X 0,Y 63.156,Z 869.21,A -85,B 0,C 180,E1 2715.012,E2 2715.012} C_VEL
LIN {X 0,Y 81.457,Z 860.457,A -85,B 0,C 180,E1 2706.085,E2 2706.085} C_VEL
LIN {X 0,Y 99.006,Z 850.724,A -85,B 0,C 180,E1 2700.858,E2 2700.858} C_VEL
LIN {X 0,Y 117.64,Z 838.687,A -85,B 0,C 180,E1 2697.079,E2 2697.079} C_VEL
LIN {X 0,Y 134.598,Z 825.967,A -85,B 0,C 180,E1 2694.553,E2 2694.553} C_VEL
LIN {X 0,Y 151.751,Z 810.979,A -85,B 0,C 180,E1 2692.6,E2 2692.6} C_VEL
LIN {X 0,Y 166.948,Z 795.456,A -85,B 0,C 180,E1 2691.205,E2 2691.205} C_VEL
LIN {X 0,Y 180.908,Z 778.95,A -85,B 0,C 180,E1 2690.136,E2 2690.136} C_VEL
LIN {X 0,Y 193.73,Z 761.36,A -85,B 0,C 180,E1 2689.293,E2 2689.293} C_VEL
LIN {X 0,Y 205.517,Z 742.353,A -85,B 0,C 180,E1 2688.623,E2 2688.623} C_VEL
LIN {X 0,Y 216,Z 721.965,A -85,B 0,C 180,E1 2688.092,E2 2688.092} C_VEL
LIN {X 0,Y 224.688,Z 701.272,A -85,B 0,C 180,E1 2687.691,E2 2687.691} C_VEL
LIN {X 0,Y 232.025,Z 679.132,A -85,B 0,C 180,E1 2687.389,E2 2687.389} C_VEL
LIN {X 0,Y 237.341,Z 657.422,A -85,B 0,C 180,E1 2687.117,E2 2687.117} C_VEL
LIN {X 0,Y 241.002,Z 634.813,A -85,B 0,C 180,E1 2686.814,E2 2686.814} C_VEL
LIN {X 0,Y 253.11,Z 538.192,A -85,B 0,C 180,E1 2685.59,E2 2685.59} C_VEL
LIN {X 0,Y 251.642,Z 535.579,A -85,B 0,C 180,E1 2680.341,E2 2680.341} C_VEL
LIN {X 0,Y 251.186,Z 537.634,A -85,B 0,C 180,E1 2675.558,E2 2675.558} C_VEL
LIN {X 0,Y 236.306,Z 647.064,A -85,B 0,C 180,E1 2674.484,E2 2674.484} C_VEL
LIN {X 0,Y 231.218,Z 670.057,A -85,B 0,C 180,E1 2674.216,E2 2674.216} C_VEL
LIN {X 0,Y 224.681,Z 691.237,A -85,B 0,C 180,E1 2673.862,E2 2673.862} C_VEL
LIN {X 0,Y 216.506,Z 711.912,A -85,B 0,C 180,E1 2673.388,E2 2673.388} C_VEL
LIN {X 0,Y 206.875,Z 731.663,A -85,B 0,C 180,E1 2672.79,E2 2672.79} C_VEL
LIN {X 0,Y 195.838,Z 750.494,A -85,B 0,C 180,E1 2672.043,E2 2672.043} C_VEL
LIN {X 0,Y 183.321,Z 768.53,A -85,B 0,C 180,E1 2671.096,E2 2671.096} C_VEL
LIN {X 0,Y 168.853,Z 786.186,A -85,B 0,C 180,E1 2669.836,E2 2669.836} C_VEL
LIN {X 0,Y 153.452,Z 802.112,A -85,B 0,C 180,E1 2668.251,E2 2668.251} C_VEL
LIN {X 0,Y 138.155,Z 815.687,A -85,B 0,C 180,E1 2666.34,E2 2666.34} C_VEL
LIN {X 0,Y 121.53,Z 828.426,A -85,B 0,C 180,E1 2663.74,E2 2663.74} C_VEL
LIN {X 0,Y 104.205,Z 839.808,A -85,B 0,C 180,E1 2660.147,E2 2660.147} C_VEL
LIN {X 0,Y 86.404,Z 849.783,A -85,B 0,C 180,E1 2654.91,E2 2654.91} C_VEL
LIN {X 0,Y 68.588,Z 858.232,A -85,B 0,C 180,E1 2646.706,E2 2646.706} C_VEL
LIN {X 0,Y 53.445,Z 864.488,A -85,B 0,C 180,E1 2634.316,E2 2634.316} C_VEL
LIN {X 0,Y 41.429,Z 869.461,A -85,B 0,C 180,E1 2612.781,E2 2612.781} C_VEL
LIN {X 0,Y 37.346,Z 872.649,A -85,B 0,C 180,E1 2584.654,E2 2584.654} C_VEL
LIN {X 0,Y 42.016,Z 874.544,A -85,B 0,C 180,E1 2556.016,E2 2556.016} C_VEL
LIN {X 0,Y 55.646,Z 875.155,A -85,B 0,C 180,E1 2534.048,E2 2534.048} C_VEL
LIN {X 0,Y 73.997,Z 874.07,A -85,B 0,C 180,E1 2521.288,E2 2521.288} C_VEL
LIN {X 0,Y 87.203,Z 872.408,A -85,B 0,C 180,E1 2515.864,E2 2515.864} C_VEL
LIN {X 0,Y 64.81,Z 878.052,A -85,B 0,C 180,E1 2506.351,E2 2506.351} C_VEL
LIN {X 0,Y 46.466,Z 881.769,A -85,B 0,C 180,E1 2489.371,E2 2489.371} C_VEL
LIN {X 0,Y 35.942,Z 883.62,A -85,B 0,C 180,E1 2460.03,E2 2460.03} C_VEL
LIN {X 0,Y 35.835,Z 883.917,A -85,B 0,C 180,E1 2431.582,E2 2431.582} C_VEL
LIN {X 0,Y 35.827,Z 883.825,A -85,B 0,C 180,E1 2428.384,E2 2428.384} C_VEL
LIN {X 0,Y 36.138,Z 881.34,A -85,B 0,C 180,E1 2400.113,E2 2400.113} C_VEL
LIN {X 0,Y 44.712,Z 877.066,A -85,B 0,C 180,E1 2374.144,E2 2374.144} C_VEL
LIN {X 0,Y 47.572,Z 875.811,A -85,B 0,C 180,E1 2369.733,E2 2369.733} C_VEL
LIN {X 0,Y 51.975,Z 873.619,A -85,B 0,C 180,E1 2362.846,E2 2362.846} C_VEL
LIN {X 0,Y 64.016,Z 866.397,A -85,B 0,C 180,E1 2346.876,E2 2346.876} C_VEL
LIN {X 0,Y 69.2,Z 863.921,A -85,B 0,C 180,E1 2343.927,E2 2343.927} C_VEL
LIN {X 0,Y 88.039,Z 854.626,A -85,B 0,C 180,E1 2338.236,E2 2338.236} C_VEL
LIN {X 0,Y 106.538,Z 843.864,A -85,B 0,C 180,E1 2334.617,E2 2334.617} C_VEL
LIN {X 0,Y 124.436,Z 831.691,A -85,B 0,C 180,E1 2332.151,E2 2332.151} C_VEL
LIN {X 0,Y 142.007,Z 817.679,A -85,B 0,C 180,E1 2330.329,E2 2330.329} C_VEL
LIN {X 0,Y 158.403,Z 802.31,A -85,B 0,C 180,E1 2328.988,E2 2328.988} C_VEL
LIN {X 0,Y 173.174,Z 786.204,A -85,B 0,C 180,E1 2328.005,E2 2328.005} C_VEL
LIN {X 0,Y 187.654,Z 767.75,A -85,B 0,C 180,E1 2327.188,E2 2327.188} C_VEL
LIN {X 0,Y 199.92,Z 749.339,A -85,B 0,C 180,E1 2326.603,E2 2326.603} C_VEL
LIN {X 0,Y 210.598,Z 730.369,A -85,B 0,C 180,E1 2326.155,E2 2326.155} C_VEL
LIN {X 0,Y 220.042,Z 709.913,A -85,B 0,C 180,E1 2325.797,E2 2325.797} C_VEL
LIN {X 0,Y 227.773,Z 689.118,A -85,B 0,C 180,E1 2325.538,E2 2325.538} C_VEL
LIN {X 0,Y 234.131,Z 666.813,A -85,B 0,C 180,E1 2325.308,E2 2325.308} C_VEL
LIN {X 0,Y 238.526,Z 644.789,A -85,B 0,C 180,E1 2325.045,E2 2325.045} C_VEL
LIN {X 0,Y 251.39,Z 545.24,A -85,B 0,C 180,E1 2323.836,E2 2323.836} C_VEL
LIN {X 0,Y 250.587,Z 543.521,A -85,B 0,C 180,E1 2320.336,E2 2320.336} C_VEL
LIN {X 0,Y 250.101,Z 544.918,A -85,B 0,C 180,E1 2317.321,E2 2317.321} C_VEL
LIN {X 0,Y 236.118,Z 647.313,A -85,B 0,C 180,E1 2316.423,E2 2316.423} C_VEL
LIN {X 0,Y 231.033,Z 670.221,A -85,B 0,C 180,E1 2316.199,E2 2316.199} C_VEL
LIN {X 0,Y 224.541,Z 691.223,A -85,B 0,C 180,E1 2315.906,E2 2315.906} C_VEL
LIN {X 0,Y 216.442,Z 711.71,A -85,B 0,C 180,E1 2315.517,E2 2315.517} C_VEL
LIN {X 0,Y 206.32,Z 732.383,A -85,B 0,C 180,E1 2314.995,E2 2314.995} C_VEL
LIN {X 0,Y 194.861,Z 751.699,A -85,B 0,C 180,E1 2314.352,E2 2314.352} C_VEL
LIN {X 0,Y 182.551,Z 769.241,A -85,B 0,C 180,E1 2313.581,E2 2313.581} C_VEL
LIN {X 0,Y 167.921,Z 786.904,A -85,B 0,C 180,E1 2312.529,E2 2312.529} C_VEL
LIN {X 0,Y 152.247,Z 802.921,A -85,B 0,C 180,E1 2311.201,E2 2311.201} C_VEL
LIN {X 0,Y 135.784,Z 817.278,A -85,B 0,C 180,E1 2309.497,E2 2309.497} C_VEL
LIN {X 0,Y 118.841,Z 829.919,A -85,B 0,C 180,E1 2307.29,E2 2307.29} C_VEL
LIN {X 0,Y 100.665,Z 841.464,A -85,B 0,C 180,E1 2304.128,E2 2304.128} C_VEL
LIN {X 0,Y 82.665,Z 851.141,A -85,B 0,C 180,E1 2299.651,E2 2299.651} C_VEL
LIN {X 0,Y 63.935,Z 859.56,A -85,B 0,C 180,E1 2292.269,E2 2292.269} C_VEL
LIN {X 0,Y 46.72,Z 866.074,A -85,B 0,C 180,E1 2279.501,E2 2279.501} C_VEL
LIN {X 0,Y 33.884,Z 870.724,A -85,B 0,C 180,E1 2256.796,E2 2256.796} C_VEL
LIN {X 0,Y 29.467,Z 873.923,A -85,B 0,C 180,E1 2221.661,E2 2221.661} C_VEL
LIN {X 0,Y 36.125,Z 875.837,A -85,B 0,C 180,E1 2187.702,E2 2187.702} C_VEL
LIN {X 0,Y 52.277,Z 876.474,A -85,B 0,C 180,E1 2166.091,E2 2166.091} C_VEL
LIN {X 0,Y 69.127,Z 875.758,A -85,B 0,C 180,E1 2156.249,E2 2156.249} C_VEL
LIN {X 0,Y 46.947,Z 879.839,A -85,B 0,C 180,E1 2143.369,E2 2143.369} C_VEL
LIN {X 0,Y 30.753,Z 882.069,A -85,B 0,C 180,E1 2115.638,E2 2115.638} C_VEL
LIN {X 0,Y 27.301,Z 882.56,A -85,B 0,C 180,E1 2078.402,E2 2078.402} C_VEL
LIN {X 0,Y 27.948,Z 882.539,A -85,B 0,C 180,E1 2069.979,E2 2069.979} C_VEL
LIN {X 0,Y 28.887,Z 879.977,A -85,B 0,C 180,E1 2033.93,E2 2033.93} C_VEL
LIN {X 0,Y 39.903,Z 875.62,A -85,B 0,C 180,E1 2005.218,E2 2005.218} C_VEL
LIN {X 0,Y 56.843,Z 869.154,A -85,B 0,C 180,E1 1989.869,E2 1989.869} C_VEL
LIN {X 0,Y 69.2,Z 863.921,A -85,B 0,C 180,E1 1983.927,E2 1983.927} C_VEL
LIN {X 0,Y 75.276,Z 860.881,A -85,B 0,C 180,E1 1980.943,E2 1980.943} C_VEL
LIN {X 0,Y 90.472,Z 851.609,A -85,B 0,C 180,E1 1972.886,E2 1972.886} C_VEL
LIN {X 0,Y 95.924,Z 848.357,A -85,B 0,C 180,E1 1971.569,E2 1971.569} C_VEL
LIN {X 0,Y 115.005,Z 836.502,A -85,B 0,C 180,E1 1969.266,E2 1969.266} C_VEL
LIN {X 0,Y 131.995,Z 824.142,A -85,B 0,C 180,E1 1967.752,E2 1967.752} C_VEL
LIN {X 0,Y 149.426,Z 809.26,A -85,B 0,C 180,E1 1966.567,E2 1966.567} C_VEL
LIN {X 0,Y 165.097,Z 793.533,A -85,B 0,C 180,E1 1965.706,E2 1965.706} C_VEL
LIN {X 0,Y 179.562,Z 776.592,A -85,B 0,C 180,E1 1965.049,E2 1965.049} C_VEL
LIN {X 0,Y 192.973,Z 758.177,A -85,B 0,C 180,E1 1964.531,E2 1964.531} C_VEL
LIN {X 0,Y 204.777,Z 739.006,A -85,B 0,C 180,E1 1964.138,E2 1964.138} C_VEL
LIN {X 0,Y 215.064,Z 718.94,A -85,B 0,C 180,E1 1963.832,E2 1963.832} C_VEL
LIN {X 0,Y 223.837,Z 697.724,A -85,B 0,C 180,E1 1963.598,E2 1963.598} C_VEL
LIN {X 0,Y 230.71,Z 676.534,A -85,B 0,C 180,E1 1963.436,E2 1963.436} C_VEL
LIN {X 0,Y 236.034,Z 654.242,A -85,B 0,C 180,E1 1963.233,E2 1963.233} C_VEL
LIN {X 0,Y 240.028,Z 628.39,A -85,B 0,C 180,E1 1962.947,E2 1962.947} C_VEL
LIN {X 0,Y 249.841,Z 552.287,A -85,B 0,C 180,E1 1962.113,E2 1962.113} C_VEL
LIN {X 0,Y 249.525,Z 551.467,A -85,B 0,C 180,E1 1960.332,E2 1960.332} C_VEL
LIN {X 0,Y 249.253,Z 552.2,A -85,B 0,C 180,E1 1959.097,E2 1959.097} C_VEL
LIN {X 0,Y 236.147,Z 647.648,A -85,B 0,C 180,E1 1958.363,E2 1958.363} C_VEL
LIN {X 0,Y 231.029,Z 670.63,A -85,B 0,C 180,E1 1958.18,E2 1958.18} C_VEL
LIN {X 0,Y 224.405,Z 691.94,A -85,B 0,C 180,E1 1957.941,E2 1957.941} C_VEL
LIN {X 0,Y 216.258,Z 712.394,A -85,B 0,C 180,E1 1957.627,E2 1957.627} C_VEL
LIN {X 0,Y 206.07,Z 733.058,A -85,B 0,C 180,E1 1957.209,E2 1957.209} C_VEL
LIN {X 0,Y 194.63,Z 752.229,A -85,B 0,C 180,E1 1956.7,E2 1956.7} C_VEL
LIN {X 0,Y 182.125,Z 769.935,A -85,B 0,C 180,E1 1956.082,E2 1956.082} C_VEL
LIN {X 0,Y 167.365,Z 787.617,A -85,B 0,C 180,E1 1955.246,E2 1955.246} C_VEL
LIN {X 0,Y 151.629,Z 803.547,A -85,B 0,C 180,E1 1954.203,E2 1954.203} C_VEL
LIN {X 0,Y 135.865,Z 817.206,A -85,B 0,C 180,E1 1952.94,E2 1952.94} C_VEL
LIN {X 0,Y 117.637,Z 830.699,A -85,B 0,C 180,E1 1951.108,E2 1951.108} C_VEL
LIN {X 0,Y 99.503,Z 842.044,A -85,B 0,C 180,E1 1948.673,E2 1948.673} C_VEL
LIN {X 0,Y 80.534,Z 852.009,A -85,B 0,C 180,E1 1945.038,E2 1945.038} C_VEL
LIN {X 0,Y 60.926,Z 860.462,A -85,B 0,C 180,E1 1939.032,E2 1939.032} C_VEL
LIN {X 0,Y 43.152,Z 866.753,A -85,B 0,C 180,E1 1928.744,E2 1928.744} C_VEL
LIN {X 0,Y 27.223,Z 871.783,A -85,B 0,C 180,E1 1904.921,E2 1904.921} C_VEL
LIN {X 0,Y 21.591,Z 875.062,A -85,B 0,C 180,E1 1859.409,E2 1859.409} C_VEL
LIN {X 0,Y 30.476,Z 877.048,A -85,B 0,C 180,E1 1817.994,E2 1817.994} C_VEL
LIN {X 0,Y 49.316,Z 877.803,A -85,B 0,C 180,E1 1797.672,E2 1797.672} C_VEL
LIN {X 0,Y 50.764,Z 877.795,A -85,B 0,C 180,E1 1796.775,E2 1796.775} C_VEL
LIN {X 0,Y 30.101,Z 880.376,A -85,B 0,C 180,E1 1778.39,E2 1778.39} C_VEL
LIN {X 0,Y 19.396,Z 881.155,A -85,B 0,C 180,E1 1734.322,E2 1734.322} C_VEL
LIN {X 0,Y 19.865,Z 881.102,A -85,B 0,C 180,E1 1709.97,E2 1709.97} C_VEL
LIN {X 0,Y 22.708,Z 878.42,A -85,B 0,C 180,E1 1661.498,E2 1661.498} C_VEL
LIN {X 0,Y 37.915,Z 873.583,A -85,B 0,C 180,E1 1632.58,E2 1632.58} C_VEL
LIN {X 0,Y 57.008,Z 866.881,A -85,B 0,C 180,E1 1620.852,E2 1620.852} C_VEL
LIN {X 0,Y 77.31,Z 858.095,A -85,B 0,C 180,E1 1614.853,E2 1614.853} C_VEL
LIN {X 0,Y 95.924,Z 848.357,A -85,B 0,C 180,E1 1611.569,E2 1611.569} C_VEL
LIN {X 0,Y 102.212,Z 844.521,A -85,B 0,C 180,E1 1610.148,E2 1610.148} C_VEL
LIN {X 0,Y 117.849,Z 833.315,A -85,B 0,C 180,E1 1605.417,E2 1605.417} C_VEL
LIN {X 0,Y 123.071,Z 829.422,A -85,B 0,C 180,E1 1604.739,E2 1604.739} C_VEL
LIN {X 0,Y 140.535,Z 815.734,A -85,B 0,C 180,E1 1603.851,E2 1603.851} C_VEL
LIN {X 0,Y 157.214,Z 800.31,A -85,B 0,C 180,E1 1603.178,E2 1603.178} C_VEL
LIN {X 0,Y 172.291,Z 783.988,A -85,B 0,C 180,E1 1602.687,E2 1602.687} C_VEL
LIN {X 0,Y 186.481,Z 765.994,A -85,B 0,C 180,E1 1602.294,E2 1602.294} C_VEL
LIN {X 0,Y 199.232,Z 746.865,A -85,B 0,C 180,E1 1602,E2 1602} C_VEL
LIN {X 0,Y 209.823,Z 727.954,A -85,B 0,C 180,E1 1601.788,E2 1601.788} C_VEL
LIN {X 0,Y 219.157,Z 707.734,A -85,B 0,C 180,E1 1601.621,E2 1601.621} C_VEL
LIN {X 0,Y 226.935,Z 686.602,A -85,B 0,C 180,E1 1601.506,E2 1601.506} C_VEL
LIN {X 0,Y 232.942,Z 665.292,A -85,B 0,C 180,E1 1601.386,E2 1601.386} C_VEL
LIN {X 0,Y 237.488,Z 642.206,A -85,B 0,C 180,E1 1601.178,E2 1601.178} C_VEL
LIN {X 0,Y 244.251,Z 591.537,A -85,B 0,C 180,E1 1600.672,E2 1600.672} C_VEL
LIN {X 0,Y 236.277,Z 648.513,A -85,B 0,C 180,E1 1600.298,E2 1600.298} C_VEL
LIN {X 0,Y 231.138,Z 671.427,A -85,B 0,C 180,E1 1600.157,E2 1600.157} C_VEL
LIN {X 0,Y 224.294,Z 693.217,A -85,B 0,C 180,E1 1599.97,E2 1599.97} C_VEL
LIN {X 0,Y 216.363,Z 712.925,A -85,B 0,C 180,E1 1599.742,E2 1599.742} C_VEL
LIN {X 0,Y 206.125,Z 733.601,A -85,B 0,C 180,E1 1599.428,E2 1599.428} C_VEL
LIN {X 0,Y 194.855,Z 752.443,A -85,B 0,C 180,E1 1599.057,E2 1599.057} C_VEL
LIN {X 0,Y 182.043,Z 770.521,A -85,B 0,C 180,E1 1598.593,E2 1598.593} C_VEL
LIN {X 0,Y 167.182,Z 788.216,A -85,B 0,C 180,E1 1597.98,E2 1597.98} C_VEL
LIN {X 0,Y 151.292,Z 804.212,A -85,B 0,C 180,E1 1597.218,E2 1597.218} C_VEL
LIN {X 0,Y 135.407,Z 817.892,A -85,B 0,C 180,E1 1596.304,E2 1596.304} C_VEL
LIN {X 0,Y 116.962,Z 831.439,A -85,B 0,C 180,E1 1594.989,E2 1594.989} C_VEL
LIN {X 0,Y 98.542,Z 842.843,A -85,B 0,C 180,E1 1593.251,E2 1593.251} C_VEL
LIN {X 0,Y 79.149,Z 852.867,A -85,B 0,C 180,E1 1590.665,E2 1590.665} C_VEL
LIN {X 0,Y 58.843,Z 861.351,A -85,B 0,C 180,E1 1586.384,E2 1586.384} C_VEL
LIN {X 0,Y 39.032,Z 867.971,A -85,B 0,C 180,E1 1578.246,E2 1578.246} C_VEL
LIN {X 0,Y 20.634,Z 873.028,A -85,B 0,C 180,E1 1555.887,E2 1555.887} C_VEL
LIN {X 0,Y 14.019,Z 876.33,A -85,B 0,C 180,E1 1490.121,E2 1490.121} C_VEL
LIN {X 0,Y 28.001,Z 878.423,A -85,B 0,C 180,E1 1441.943,E2 1441.943} C_VEL
LIN {X 0,Y 31.948,Z 878.752,A -85,B 0,C 180,E1 1437.722,E2 1437.722} C_VEL
LIN {X 0,Y 13.321,Z 879.728,A -85,B 0,C 180,E1 1398.572,E2 1398.572} C_VEL
LIN {X 0,Y 11.735,Z 879.638,A -85,B 0,C 180,E1 1349.95,E2 1349.95} C_VEL
LIN {X 0,Y 18.289,Z 876.837,A -85,B 0,C 180,E1 1281.577,E2 1281.577} C_VEL
LIN {X 0,Y 37.005,Z 871.795,A -85,B 0,C 180,E1 1259.723,E2 1259.723} C_VEL
LIN {X 0,Y 56.474,Z 865.278,A -85,B 0,C 180,E1 1252.587,E2 1252.587} C_VEL
LIN {X 0,Y 77.169,Z 856.54,A -85,B 0,C 180,E1 1248.796,E2 1248.796} C_VEL
LIN {X 0,Y 96.607,Z 846.428,A -85,B 0,C 180,E1 1246.649,E2 1246.649} C_VEL
LIN {X 0,Y 115.85,Z 834.458,A -85,B 0,C 180,E1 1245.174,E2 1245.174} C_VEL
LIN {X 0,Y 123.071,Z 829.422,A -85,B 0,C 180,E1 1244.739,E2 1244.739} C_VEL
LIN {X 0,Y 129.029,Z 824.853,A -85,B 0,C 180,E1 1243.967,E2 1243.967} C_VEL
LIN {X 0,Y 143.178,Z 812.429,A -85,B 0,C 180,E1 1240.926,E2 1240.926} C_VEL
LIN {X 0,Y 148.896,Z 807.253,A -85,B 0,C 180,E1 1240.414,E2 1240.414} C_VEL
LIN {X 0,Y 153.434,Z 802.91,A -85,B 0,C 180,E1 1240.305,E2 1240.305} C_VEL
LIN {X 0,Y 136.449,Z 817.734,A -85,B 0,C 180,E1 1239.72,E2 1239.72} C_VEL
LIN {X 0,Y 118.895,Z 830.779,A -85,B 0,C 180,E1 1238.993,E2 1238.993} C_VEL
LIN {X 0,Y 100.289,Z 842.452,A -85,B 0,C 180,E1 1238.015,E2 1238.015} C_VEL
LIN {X 0,Y 80.617,Z 852.651,A -85,B 0,C 180,E1 1236.623,E2 1236.623} C_VEL
LIN {X 0,Y 60.384,Z 861.219,A -85,B 0,C 180,E1 1234.504,E2 1234.504} C_VEL
LIN {X 0,Y 39.093,Z 868.355,A -85,B 0,C 180,E1 1230.442,E2 1230.442} C_VEL
LIN {X 0,Y 19.469,Z 873.44,A -85,B 0,C 180,E1 1220.433,E2 1220.433} C_VEL
LIN {X 0,Y 5.658,Z 876.902,A -85,B 0,C 180,E1 1138.109,E2 1138.109} C_VEL
LIN {X 0,Y 12.141,Z 878.279,A -85,B 0,C 180,E1 1080.861,E2 1080.861} C_VEL
LIN {X 0,Y 3.554,Z 878.163,A -85,B 0,C 180,E1 989.834,E2 989.834} C_VEL
LIN {X 0,Y 17.085,Z 875.248,A -85,B 0,C 180,E1 894.561,E2 894.561} C_VEL
LIN {X 0,Y 36.942,Z 870.285,A -85,B 0,C 180,E1 887.064,E2 887.064} C_VEL
LIN {X 0,Y 58.191,Z 863.219,A -85,B 0,C 180,E1 884.232,E2 884.232} C_VEL
LIN {X 0,Y 78.531,Z 854.63,A -85,B 0,C 180,E1 882.751,E2 882.751} C_VEL
LIN {X 0,Y 97.876,Z 844.539,A -85,B 0,C 180,E1 881.831,E2 881.831} C_VEL
LIN {X 0,Y 116.194,Z 833.074,A -85,B 0,C 180,E1 881.198,E2 881.198} C_VEL
LIN {X 0,Y 134.539,Z 819.52,A -85,B 0,C 180,E1 880.716,E2 880.716} C_VEL
LIN {X 0,Y 148.896,Z 807.253,A -85,B 0,C 180,E1 880.414,E2 880.414} C_VEL
LIN {X 0,Y 152.216,Z 808.752,A -85,B 0,C 180,E1 880.351,E2 880.351} C_VEL
LIN {X 0,Y 152.216,Z 951,A -85,B 0,C 180,E1 880.351,E2 880.351} C_VEL
LIN {X 0,Y 152.216,Z 951,A -85,B 0,C 180,E1 880.351,E2 880.351}

QRS_NEXT_CUT()

QRS_NEXT()
QRS_HOME()

END
